PROGRAM P2_DriveLoad
VAR




	
// Loads CMP80M & M700 initial parameters.
	//CMP80M	: INT;
	//netId	: INT;
	//port	: INT;
	//bLoadParameters_Done: BOOL;
	

	
	
END_VAR



GVL_Index.Decel_For_DeadMan := 10000;
GVL_Index.Decel_For_Estop := 20000;
GVL_Motion.rHoist_MaxVelocity := 1000;
//GVL_Speeds.rAccel_With_MinLoad :=1000;
//GVL_Speeds.rDecel_With_MinLoad := 1000;
//nMotion_Command := 10;
KidAxis.modeAcc := 800;
GVL_Motion.lrDistance_1_Motor_Rev := 300;
//GVL_Motion.rMotor_GearRatio := 1;
//GVL_Motion.tMotorBrake_Delay := T#15S;
//GVL_Motion.lrDrum_Diameter := 300;
GVL_Motion.lrEncoder_ScalingNum := 0.00092327;
bLoadParameters_Done				:=	TRUE;

(*
//*****************************************************************Notes**********************************************************\\

  	The P_Drive_Verification program confirms that the drive parameters are set according to the motor that it is currently set up as.
	This will prevent any motion from occuring and throw an error if the parameters aren't set correctly.

  
  
//*****************************************************************Revs**********************************************************\\
   (          who            )(    Date    ) (   Rev     ) (								Disc						)
     Brent Miller			 	2016.04.08		0.00.01		Initial Code.
     		 								 				
	 						
	
//*****************************************************************Code**********************************************************\\


//	Has Drive already been verified?

IF NOT GVL_Modes.bDrive_Verified	THEN
		
	//This code will run if drive settings have not been verified
	//Will return a True value to bDrive_Verified
	//The HMI will need to load settings by setting a value of 1-100 in the Motor_Load_Parameters tag
	CASE GVL_HMI.Motor_Load_Parameters OF
		
	0:
		GVL_HMI.Motor_Load_Parameters	:= 1;
		A3_LoadParameters_Tracking();
		IF bLoadParameters_Done THEN
			GVL_Modes.bDrive_Verified := TRUE;
		END_IF
		
	1:
		A1_LoadParameters_ZipLift_CMP80M();
	//	GVL_HMI.Motor_Load_Parameters	:= 0;
		IF bLoadParameters_Done THEN
			GVL_Modes.bDrive_Verified := TRUE;
		END_IF
		
	2:
		A2_LoadParameters_ZipLift_FM050();	//
	//	GVL_HMI.Motor_Load_Parameters	:= 0;
		IF bLoadParameters_Done THEN
			GVL_Modes.bDrive_Verified := TRUE;
		END_IF
		
	ELSE	//if not any of the values listed above in Case statement then run this code
		//Figure out a way to trip the drive or prevent system from operating if bDrive_Verified = FALSE
		//pprasinos 6/9/2017 GVL_HMI.Drive_Status_Trip 	:=	E_Custom_Trip_Codes.System_Model_Unknown;
		
		//After the trip is Ack. then this needs to clear and set back to "OK"
		//pprasinos 6/9/2017 GVL_HMI.Drive_Status_Trip	:=	E_Custom_Trip_Codes.OK;
	
		
	END_CASE;
	
	
	
END_IF




*)

ACTION A1_LoadParameters_ZipLift_CMP80M:

GVL_Index.Decel_For_DeadMan := 10000;
GVL_Index.Decel_For_Estop := 20000;
GVL_Motion.rHoist_MaxVelocity := 1500;
//GVL_Speeds.rAccel_With_MinLoad :=1000;
//GVL_Speeds.rDecel_With_MinLoad := 1000;
//nMotion_Command := 10;
KidAxis.modeAcc := 1200;
GVL_Motion.lrDistance_1_Motor_Rev := 300;
//GVL_Motion.rMotor_GearRatio := 1;
//GVL_Motion.tMotorBrake_Delay := T#15S;
//GVL_Motion.lrDrum_Diameter := 300;
GVL_Motion.lrEncoder_ScalingNum := 0.00092327;
bLoadParameters_Done				:=	TRUE;
END_ACTION

END_PROGRAM

(* stored: Version 1.1.0.1, ProductVersion 3.1.4022.7
   POU P2_DriveLoad: Id {d95ea949-7ad0-4176-be6d-d221148a2996}, SpecialFunc None
   Action A1_LoadParameters_ZipLift_CMP80M: Id {f2719792-c7b1-4f91-81ed-b3619ef7c9fa} *)
